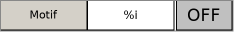
VISUALIZATION VISU_BAL_MANU  // 234x32
VAR_IN_OUT
	m_Input_BAL: BLOCK_TELEMARK_DIGITAL_SWEEP;
END_VAR
    Rectangle (87,0 87x30), "%i", text variable: m_Input_BAL.PRM_NbBal, input disabled if: NOT (Global_Variables.PRG_USER.ACTU_USER.FONCTION_SA AND NOT MACHINE.STATE_PROD)
        OnMouseClick: write the text variable via VisuDialogs.Numpad, min 1, max 8
    RoundedRectangle (176,0 56x30), "ON", invisible if: NOT m_Input_BAL.STATE_ON
    RoundedRectangle (176,0 56x30), "OFF", invisible if: NOT m_Input_BAL.STATE_OFF
    Rectangle (0,0 87x30), "Motif"
END_VISUALIZATION

(* stored: Version 1.1.0.1, ProductVersion 3.1.4024.10
   Visu VISU_BAL_MANU: Id {fffe2c5e-d474-4f5b-9ea2-34d3de61c61b} *)
